PROGRAM Test
VAR
    fbCallCtrlTest: FB_InvocationControl_Test;
    fbObserverTest: FB_ObserverPattern_Test;
END_VAR

TcUnit.RUN();

END_PROGRAM

(* stored: Version 1.1.0.1, ProductVersion 3.1.4024.12
   POU Test: Id {6350dc1d-88ea-43c9-9a34-501ba75d0b98}, SpecialFunc None *)
